TYPE HMINumericalInputLineInterface :
STRUCT
	CaptionDescription	:	STRING;
	UnitInput	:	STRING;
	ValueInput	:	REAL;
	IsEnabledInput	:	BOOL;
END_STRUCT
END_TYPE

(* stored: Version 1.1.0.1
   DUT HMINumericalInputLineInterface: Id {5826f568-2635-4280-a5f8-e95b72d53c03} *)
